(* IEC 61131-3 sources: Industry-PLC-LLM/data/PLCBEAD_repo/PLCBEAD_PLCEmbed-main/PLC-BEAD/Source/GEB/HOUR, 1 file *)

(* ---- HOUR.ST ---- *)
FUNCTION HOUR:INT
	VAR_INPUT
		ITOD :	UDINT;
	END_VAR
	HOUR := UDINT_TO_INT(ITOD / UDINT#3600000);
END_FUNCTION

PROGRAM program0
  VAR
	  ITOD :	UDINT;
    CEIL5_OUT : INT;
  END_VAR

  CEIL5_OUT := HOUR(ITOD);
END_PROGRAM
